TYPE ST_ActuatorInputs :
STRUCT
	Advanced  AT%I* : BOOL;
	Retracted AT%I* : BOOL;
END_STRUCT
END_TYPE

(* stored: Version 1.1.0.1, ProductVersion 3.1.4024.12
   DUT ST_ActuatorInputs: Id {48b4370c-9568-47b5-828a-80e00ef868b9} *)
